TYPE T_MioSysTimes : ARRAY [0 .. GVL.cTimeBufferDepth] OF ARRAY [GVL.cMio0 .. GVL.cMio1] OF ULINT; END_TYPE

(* stored: Version 1.1.0.1, ProductVersion 3.1.4022.18
   DUT T_MioSysTimes: Id {421feef3-879a-4082-9c7a-56b0d93ff5bd} *)
